{attribute 'GeneratedUsingTerminal: EL6090-0000-0016'}
{attribute addProperty BoxType "EL6090-0000-0016"}
{attribute addProperty Id "EtcSlaveTerminalBaseDIS_InputsAT %I*DIS_Inputs_E0E384E36DIS_OutputsAT %Q*DIS_Outputs_6C9BFFEE4WcStateAT %I*WcState_9091E0EB2InfoDataAT %I*InfoData_32EB74EA10"}
{attribute addProperty CRC "467352780"}
{attribute addProperty Size "22"}
TYPE EL6090_1BDB3CCC EXTENDS EtcSlaveTerminalBase :
STRUCT
	{attribute addProperty Name "DIS_Inputs"}
	DIS_Inputs : DIS_Inputs_E0E384E3;
	{attribute addProperty Name "DIS_Outputs"}
	DIS_Outputs : DIS_Outputs_6C9BFFEE;
	{attribute addProperty Name "WcState"}
	WcState : WcState_9091E0EB;
	{attribute addProperty Name "InfoData"}
	InfoData : InfoData_32EB74EA;
END_STRUCT
END_TYPE

(* stored: Version 1.2.0.0, ProductVersion 3.1.4024.9
   DUT EL6090_1BDB3CCC: Id {f4703ea9-9b7c-4974-9e2e-be2351dbeae2} *)
